# EPICS substitutions: src/iocdoc/testfiles/iocBoot/ioc495idc/templates/filter.substitutions
# filter.substitutions

file "$(OPTICS)/databases/filterBladeNoSensor.db" {
  pattern
  {P,      R,        N,   DESC,           OUT                  OUT_STRING,  IN_STRING}
  {495idc:,   filter:,  1,   "Filter 1",     "495idc:9440:1:bo_12.VAL",   "0",       "1"}
  {495idc:,   filter:,  2,   "Filter 2",     "495idc:9440:1:bo_13.VAL",   "0",       "1"}
  {495idc:,   filter:,  3,   "Filter 3",     "495idc:9440:1:bo_14.VAL",   "0",       "1"}
  {495idc:,   filter:,  4,   "Filter 4",     "495idc:9440:1:bo_15.VAL",   "0",       "1"}
}

file "$(OPTICS)/databases/filterDrive.db" {
  {P="495idc:", R="filter:", DESC="Filters", KEV="IDus:Energy"}
}
